{attribute 'qualified_only'}
{attribute 'strict'}
{attribute 'to_string'}
TYPE E_NORMAL_CAM_HANDLER_SEQ_STEPS :
(
	INIT := 0,

	UNDER_LIGHT_TEST_ENABLE_LIGHT,
	UNDER_LIGHT_TEST_IMAGE_ACQUIRE,
	UNDER_LIGHT_TEST_IMAGE_PROCESSING,
	UNDER_LIGHT_TEST_OK,
	UNDER_LIGHT_TEST_FAILED,

	LASER_LIGHT_TEST_ENABLE_LIGHT,
	LASER_LIGHT_TEST_IMAGE_ACQUIRE,
	LASER_LIGHT_TEST_IMAGE_PROCESSING,
	LASER_LIGHT_TEST_OK,
	LASER_LIGHT_TEST_FAILED,
	
	COUPLER_DETECT_ENABLE_LIGHT,
	COUPLER_DETECT_IMAGE_ACQUIRE,
	COUPLER_DETECT_IMAGE_PROCESSING,
	COUPLER_DETECT_DONE,
	COUPLER_DETECT_FAILED,

	MIRROR_DETECT_ENABLE_LIGHT,
	MIRROR_DETECT_IMAGE_ACQUIRE,
	MIRROR_DETECT_IMAGE_PROCESSING,
	MIRROR_DETECT_DONE,
	MIRROR_DETECT_FAILED,
	
	
	END
);
END_TYPE

(* stored: Version 1.1.0.1
   DUT E_NORMAL_CAM_HANDLER_SEQ_STEPS: Id {d91b5ded-ed84-4af9-8457-ad0ed6809423} *)
